Yaskawa INFORM job: h_profile_raised_05_05_2024.JBI

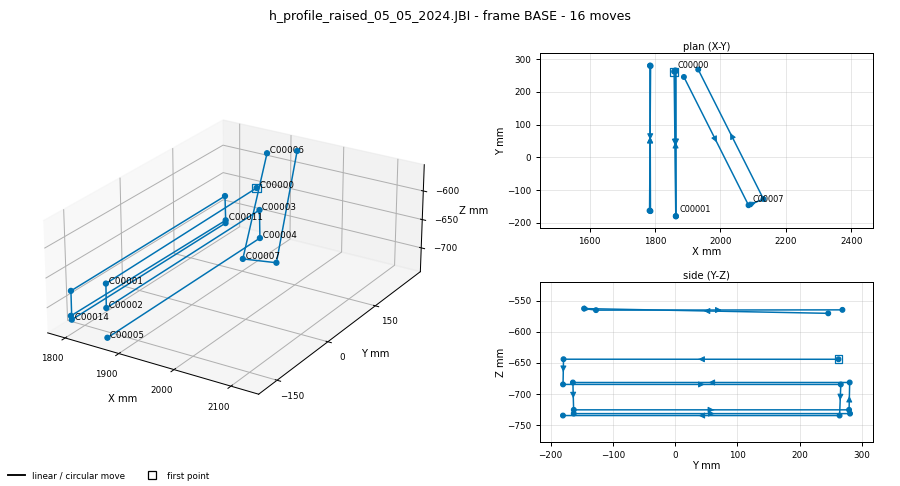
[picture p0: tool path of h_profile_raised_05_05_2024.JBI in frame BASE, 16 of 20 moves have a stored position in this frame; points joined in program order, loops and branches not executed]
/JOB
//NAME h_profile_raised_05_05_2024
//POS
///NPOS 16,0,16,0,0,0
///TOOL 0
///POSTYPE BASE
///RECTAN
///RCONF 0,0,0,0,0,0,0,0,0,0,0,0,0,0,0,0,0,0,0,0,0,0,0,0
C00000=1858.269929,262.432458,-644.043585,-5.000000,-89.321707,-175.000000
C00001=1863.332923,-179.315309,-643.952779,-5.000000,-89.321707,-175.000000
C00002=1863.471560,-180.108075,-684.430218,-5.000000,-89.321707,-175.000000
C00003=1861.787021,266.105399,-684.481339,-5.000000,-89.321707,-175.000000
C00004=1864.044994,264.151148,-734.457975,-5.000000,-89.321707,-175.000000
C00005=1864.066543,-180.213183,-734.426671,180.000000,-60.000000,0.000000
C00006=1888.191736,245.926207,-570.248950,175.000000,-5.000000,5.000000
C00007=2085.813441,-146.283237,-562.610984,175.000000,-5.000000,5.000000
C00008=2131.363160,-127.143894,-565.129984,175.000000,-5.000000,5.000000
C00009=1931.915457,268.689510,-564.663984,175.000000,-5.000000,5.000000
C00010=1783.169477,-162.799598,-725.255689,175.000000,-89.580176,-5.000000
C00011=1786.390552,279.400469,-725.259990,175.000000,-89.580176,-5.000000
C00012=1784.549773,280.371693,-681.316159,175.000000,-89.580176,-5.000000
C00013=1785.965809,-164.262339,-681.345942,175.000000,-89.580176,-5.000000
C00014=1784.739402,-162.918719,-731.338239,175.000000,-89.580176,-5.000000
C00015=1785.106211,280.928255,-731.321554,180.000000,-60.000000,0.000000
///POSTYPE PULSE
///PULSE
EC00000=183296.0
EC00001=183296.0
EC00002=183296.0
EC00003=183296.0
EC00004=183296.0
EC00005=183296.0
EC00006=211968.0
EC00007=211968.0
EC00008=211968.0
EC00009=211968.0
EC00010=367616.0
EC00011=367616.0
EC00012=367616.0
EC00013=367616.0
EC00014=367616.0
EC00015=367616.0
//INST
///DATE 2023/05/05 11:11
///ATTR SC,RW,RJ
////FRAME BASE
///GROUP1 RB1,ST1
NOP
MOVJ P009 EX000 VJ=15.00
MOVJ C00000 EC00000 VJ=15.0
CALL JOB:SPYON
MOVL C00001 EC00001 V=150.0
MOVL C00002 EC00002 V=150.0
MOVL C00003 EC00003 V=150.0
MOVL C00004 EC00004 V=150.0
MOVL C00005 EC00005 V=150.0
CALL JOB:SPYOF
MOVJ P009 VJ=15.00
MOVJ C00006 EC00006 VJ=15.0
CALL JOB:SPYON
MOVL C00007 EC00007 V=150.0
MOVL C00008 EC00008 V=150.0
MOVL C00009 EC00009 V=150.0
CALL JOB:SPYOF
MOVJ P009 VJ=15.00
MOVJ C00010 EC00010 VJ=15.0
CALL JOB:SPYON
MOVL C00011 EC00011 V=150.0
MOVL C00012 EC00012 V=150.0
MOVL C00013 EC00013 V=150.0
MOVL C00014 EC00014 V=150.0
MOVL C00015 EC00015 V=150.0
CALL JOB:SPYOF
MOVJ P009 VJ=15.00
END
